// TIA Portal project "Zadanie_Final" (V14)

(* hardware
DEVICE "S7-1200 station_1"  S7-1200 Station
   slot 0: "Rack_0"  S7-1200 Rack  Rack  V1.0
   slot 1: "PLC_1"  CPU 1214C DC/DC/DC  6ES7 214-1AG40-0XB0  V4.2
*)

// ===== PLC "PLC_1"  CPU 1214C DC/DC/DC =====

VAR_GLOBAL   // PLC tag table "Default tag table"
   "Reset" AT %M0.0 : Bool;
   "Load" AT %M0.1 : Bool;
   "UnLoad" AT %M0.2 : Bool;
   "Min_A" AT %M0.3 : Bool;
   "Min_B" AT %M0.4 : Bool;
   "Min_C" AT %M0.5 : Bool;
   "RozkZal_A" AT %M0.6 : Bool;
   "RozkZal_B" AT %M0.7 : Bool;
   "RozkZal_C" AT %M1.0 : Bool;
   "Pauza_A" AT %M1.1 : Bool;
   "Pauza_B" AT %M1.2 : Bool;
   "Pauza_C" AT %M1.3 : Bool;
   "Praca_A" AT %M1.4 : Bool;
   "Praca_B" AT %M1.5 : Bool;
   "Praca_C" AT %M1.6 : Bool;
   "Poziom_A" AT %MD100 : Real;
   "Poziom_B" AT %MD104 : Real;
   "Poziom_C" AT %MD108 : Real;
   "Masa_A" AT %MD116 : Real;
   "Masa_B" AT %MD120 : Real;
   "Masa_C" AT %MD124 : Real;
   "Masa_S" AT %MD128 : Real;
   "Pakt_A" AT %MD132 : Real;
   "Pakt_B" AT %MD136 : Real;
   "Pakt_C" AT %MD140 : Real;
   "MasaZad_A" AT %MD144 : Real;
   "MasaZad_B" AT %MD148 : Real;
   "MasaZad_C" AT %MD152 : Real;
   "Licz_Cykle" AT %MD156 : DInt;
END_VAR

// folder: System blocks/Program resources

DATA_BLOCK "LiczZal_A"   // DB1
{ S7_Optimized_Access := 'TRUE' }
AUTHOR : Simatic
FAMILY : IEC
NAME : CNTR
VERSION : 1.0
// stored: InstanceOfName IEC_COUNTER
"IEC_COUNTER"
BEGIN
END_DATA_BLOCK

DATA_BLOCK "LiczZal_B"   // DB2
{ S7_Optimized_Access := 'TRUE' }
AUTHOR : Simatic
FAMILY : IEC
NAME : CNTR
VERSION : 1.0
// stored: InstanceOfName IEC_COUNTER
"IEC_COUNTER"
BEGIN
END_DATA_BLOCK

DATA_BLOCK "LiczZal_C"   // DB3
{ S7_Optimized_Access := 'TRUE' }
AUTHOR : Simatic
FAMILY : IEC
NAME : CNTR
VERSION : 1.0
// stored: InstanceOfName IEC_COUNTER
"IEC_COUNTER"
BEGIN
END_DATA_BLOCK

DATA_BLOCK "Licz_Load"   // DB4
{ S7_Optimized_Access := 'TRUE' }
AUTHOR : Simatic
FAMILY : IEC
NAME : CNTR
VERSION : 1.0
// stored: InstanceOfName IEC_COUNTER
"IEC_COUNTER"
BEGIN
END_DATA_BLOCK

// folder: (top level)

FUNCTION "Zadanie_Final" : Void   // FC10, LAD
TITLE = Zadanie finałowe
{ S7_Optimized_Access := 'TRUE' }
VERSION : 0.1
// Proszę skorzystać z zadeklarowanych zmiennych w tablicy symboli oraz stałych wewnątrz tej funkcji. W razie potrzeby można użyć dodatkowych zmiennych.
// Szablon rozwiązania został przedstawiony w formie poniższych Networków, które trzeba zaprogramować. W razie konieczności można stworzyć własne.
// Sprawdzenia poprawności można dokonać w tablicy "watch" o nazwie "Sprawdzenie" ustawiając zmienną "Load"=1. Ponowne uruchomienie po użyciu funkcji "Reset"=1.
   VAR CONSTANT
      q_A : Real := 4.0;   // Prędkość dozowania ze zb. A
      q_B : Real := 8.0;   // Prędkość dozowania ze zb. B
      q_C : Real := 12.0;   // Prędkość dozowania ze zb. C
      q_M : Real := 15.0;   // Prędkość dozowania ze zb. M
      max_A : Real := 2500.0;   // Masa początkowa zb. A
      max_B : Real := 2500.0;   // Masa początkowa zb. B
      max_C : Real := 9000.0;   // Masa początkowa zb. C
      Lmin : Real := 12.0;   // Poziom minimalny w zb. A,B,C
      Mmax : Real := 3800.0;   // Maksymalna masa w zb. M
      Mmin : Real := 12.0;   // Minimalna masa w zb. M
      P_A : Real := 0.15;   // Stężenie dla surowca A
      P_B : Real := 0.2;   // Stężenie dla surowca B
      P_C : Real := 0.65;   // Stężenie dla surowca C
   END_VAR
BEGIN

REGION Network 1: Reset - przywrócenie nastaw początkowych
END_REGION

REGION Network 2: Start napełniania
END_REGION

REGION Network 3: Zbiornik A - symulacja poziomu
END_REGION

REGION Network 4: Zbiornik A - kalkulacja zadanej masy
END_REGION

REGION Network 5: Zbiornik A - aktualne stężenie
END_REGION

REGION Network 6: Zbiornik B - symulacja poziomu
END_REGION

REGION Network 7: Zbiornik B - kalkulacja zadanej masy
END_REGION

REGION Network 8: Zbiornik B - aktualne stężenie
END_REGION

REGION Network 9: Zbiornik C - symulacja poziomu
END_REGION

REGION Network 10: Zbiornik C - kalkulacja zadanej masy
END_REGION

REGION Network 11: Zbiornik C - aktualne stężenie
END_REGION

REGION Network 12: Aktualna sumaryczna masa w zbiorniku
END_REGION

REGION Network 13: Liczniki: załączeń (A,B,C), załadunku zbiornika oraz liczba wszystkich cykli
END_REGION

REGION Network 14: Start opróżniania
END_REGION

REGION Network 15: Symulacja opróżniania
END_REGION

REGION Network 16: Stop opróźniania
END_REGION

REGION Network 17: Koniec całego procesu napełniania
END_REGION
END_FUNCTION

ORGANIZATION_BLOCK "Main"   // OB1, LAD, ProgramCycle
TITLE = "Main Program Sweep (Cycle)"
{ S7_Optimized_Access := 'TRUE' }
VERSION : 0.1
   VAR_INPUT
      Initial_Call : Bool;   // Initial call of this OB
      Remanence : Bool;   // =True, if remanent data are available
   END_VAR
   VAR_TEMP
      zadanie : UInt;
      end : Bool;
   END_VAR
BEGIN
END_ORGANIZATION_BLOCK

ORGANIZATION_BLOCK "Cyclic"   // OB30, LAD, CyclicInterrupt
{ S7_Optimized_Access := 'TRUE' }
VERSION : 0.1
   VAR_INPUT
      Initial_Call : Bool;   // Initial call of this OB
      Event_Count : Int;   // Events discarded
   END_VAR
BEGIN

REGION Network 1
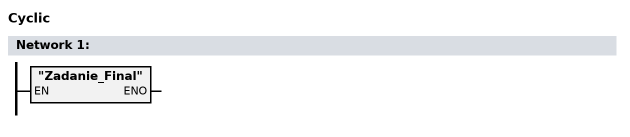
   RUNG wire#powerrail
      "Zadanie_Final"()
   END_RUNG
   // the same network as SCL:
   "Zadanie_Final"();
END_REGION
END_ORGANIZATION_BLOCK